Universal Robots PolyScope program: _adminCG-AssembleAToB.urp

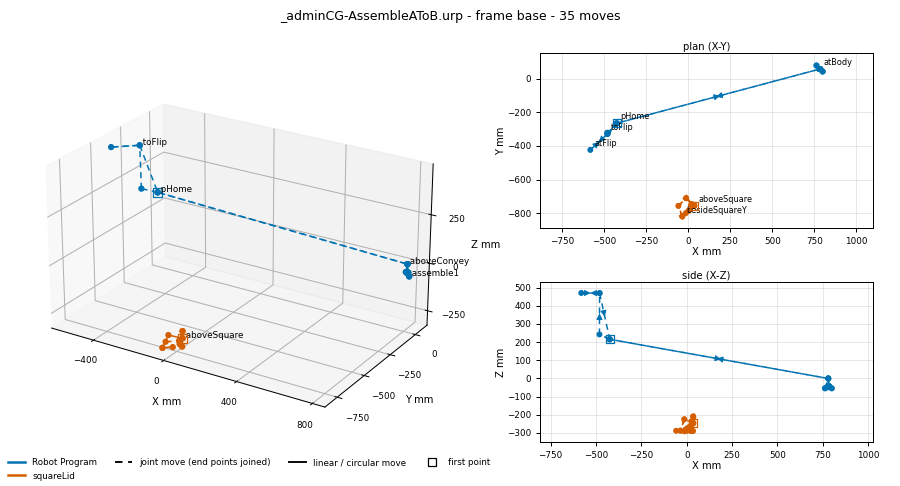
[picture p0: tool path of _adminCG-AssembleAToB.urp in frame base, 35 of 35 moves have a stored position in this frame; points joined in program order, loops and branches not executed]
Program _adminCG-AssembleAToB (installation=admin directory=/programs/WED_9AM createdIn=3.15.8.106339 lastSavedIn=3.15.8.106339 robotSerialNumber=2015350925)
Calibrated DH parameters: a=[0.000202, -0.047961, -0.392055, -0.000001, 0.000007, 0]; d=[0.089082, 828.736652, -823.627268, -4.999465, 0.094767, 0.082274]; alpha=[1.570325, 0.00051, -0.003464, 1.570175, -1.569769, 0]; deltaTheta=[0.000028, 1.457808, -1.502844, -6.238105, -6.283148, -0.000082]
Robot Program (runOnlyOnce=true)
  Set DigitalOutput pin=digital_out[0]; digitalValue=0
  MoveJ speed 60 deg/s, acceleration 80 deg/s^2 (useActiveTCP=true)
    Waypoint pHome: TCP in base x=-424.538 y=-265.05 z=215.597 mm, rx=-1.1995 ry=-2.8939 rz=-0.0048 rad; joints [224.997, -90.008, -90.005, -90.013, 89.259, -0.018] deg; flange x=-423.012 y=-266.393 z=431.487 mm, rx=-1.1995 ry=-2.8939 rz=-0.0048 rad
    Call _adminLinearIndex5
    Waypoint backUpFromFlip: TCP in base x=-481.215 y=-321.291 z=242.418 mm, rx=1.2187 ry=2.8869 rz=0.0126 rad; joints [224.559, -101.635, -73.028, -95.999, 90.041, 0.305] deg; flange x=-483.467 y=-322.229 z=458.304 mm, rx=1.2187 ry=2.8869 rz=0.0126 rad
  MoveJ speed 60 deg/s, acceleration 80 deg/s^2 (useActiveTCP=true)
    Waypoint toFlip: TCP in base x=-480.325 y=-329.398 z=470.329 mm, rx=0.0018 ry=0.0011 rz=-0.7778 rad; joints [225.307, -119.466, -107.5, -43.047, 269.775, 0.334] deg; flange x=-480.398 y=-328.953 z=254.429 mm, rx=0.0018 ry=0.0011 rz=-0.7778 rad
    Waypoint atFlip: TCP in base x=-581.465 y=-423.657 z=471.291 mm, rx=0.0073 ry=-0.0016 rz=-0.785 rad; joints [224.868, -133.376, -81.455, -55.525, 269.773, 0.333] deg; flange x=-580.559 y=-422.358 z=255.397 mm, rx=0.0073 ry=-0.0016 rz=-0.785 rad
    Set DigitalOutput pin=digital_out[0]; digitalValue=1
    Wait Sleep waitTime=1
    Set DigitalOutput pin=digital_out[2]; digitalValue=0
    Wait Sleep waitTime=1
    Waypoint toFlip: TCP in base x=-480.325 y=-329.398 z=470.329 mm, rx=0.0018 ry=0.0011 rz=-0.7778 rad; joints [225.307, -119.466, -107.5, -43.047, 269.775, 0.334] deg; flange x=-480.398 y=-328.953 z=254.429 mm, rx=0.0018 ry=0.0011 rz=-0.7778 rad
    Call _adminLinearIndex3
    Call squareLid
  MoveJ speed 60 deg/s, acceleration 80 deg/s^2 (useActiveTCP=true)
    Waypoint pHome: TCP in base x=-424.538 y=-265.05 z=215.597 mm, rx=-1.1995 ry=-2.8939 rz=-0.0048 rad; joints [224.997, -90.008, -90.005, -90.013, 89.259, -0.018] deg; flange x=-423.012 y=-266.393 z=431.487 mm, rx=-1.1995 ry=-2.8939 rz=-0.0048 rad
    Call _adminLinearIndex2
    Waypoint aboveConvey: TCP in base x=780.769 y=56.622 z=-0.465 mm, rx=1.1372 ry=-2.8707 rz=0.041 rad; joints [12.999, -136.609, -54.995, -81.263, 87.848, 59.736] deg; flange x=789.407 y=66.208 z=215.049 mm, rx=1.1372 ry=-2.8707 rz=0.041 rad
    Waypoint rotateConvey: TCP in base x=780.784 y=56.567 z=-0.471 mm, rx=2.895 ry=1.1467 rz=-0.0834 rad; joints [12.996, -136.61, -54.995, -81.26, 87.846, 239.737] deg; flange x=789.416 y=66.159 z=215.043 mm, rx=2.895 ry=1.1467 rz=-0.0834 rad
    Waypoint atBody: TCP in base x=780.781 y=56.499 z=-48.623 mm, rx=2.895 ry=1.1466 rz=-0.0836 rad; joints [12.996, -138.549, -58.718, -75.603, 87.846, 239.721] deg; flange x=789.426 y=66.117 z=166.89 mm, rx=2.895 ry=1.1466 rz=-0.0836 rad
    Wait Sleep waitTime=1
    Set DigitalOutput pin=digital_out[0]; digitalValue=0
    Wait Sleep waitTime=1
    Waypoint aboveConvey: TCP in base x=780.769 y=56.622 z=-0.465 mm, rx=1.1372 ry=-2.8707 rz=0.041 rad; joints [12.999, -136.609, -54.995, -81.263, 87.848, 59.736] deg; flange x=789.407 y=66.208 z=215.049 mm, rx=1.1372 ry=-2.8707 rz=0.041 rad
    Set DigitalOutput pin=digital_out[0]; digitalValue=1
    Waypoint abovePress: TCP in base x=785.714 y=57.816 z=-43.706 mm, rx=1.1164 ry=-2.8991 rz=0.0376 rad; joints [12.888, -138.367, -58.524, -74.941, 88.163, 60.68] deg; flange x=790.834 y=65.386 z=172.001 mm, rx=1.1164 ry=-2.8991 rz=0.0376 rad
  If force()≤65 (checkContinuously=true)
    MoveL speed 50 mm/s, acceleration 100 mm/s^2 (useActiveTCP=true) feature=Base
      Waypoint assemble1: TCP in base x=799.867 y=42.231 z=-54.523 mm, rx=1.1163 ry=-2.8991 rz=0.0375 rad; joints [11.574, -140.879, -55.504, -75.412, 88.126, 59.369] deg; flange x=805.001 y=49.793 z=161.183 mm, rx=1.1163 ry=-2.8991 rz=0.0375 rad
  MoveJ speed 60 deg/s, acceleration 80 deg/s^2 (useActiveTCP=true)
    Waypoint abovePress: TCP in base x=785.714 y=57.816 z=-43.706 mm, rx=1.1164 ry=-2.8991 rz=0.0376 rad; joints [12.888, -138.367, -58.524, -74.941, 88.163, 60.68] deg; flange x=790.834 y=65.386 z=172.001 mm, rx=1.1164 ry=-2.8991 rz=0.0376 rad
  If force()≤65 (checkContinuously=true)
    MoveL speed 50 mm/s, acceleration 100 mm/s^2 (useActiveTCP=true) feature=Base
      Waypoint assemble2: TCP in base x=763.064 y=78.057 z=-54.537 mm, rx=1.1164 ry=-2.8989 rz=0.0377 rad; joints [14.737, -135.9, -64.716, -71.278, 88.219, 62.516] deg; flange x=768.213 y=85.654 z=161.168 mm, rx=1.1164 ry=-2.8989 rz=0.0377 rad
  MoveJ speed 60 deg/s, acceleration 80 deg/s^2 (useActiveTCP=true)
    Waypoint abovePress: TCP in base x=785.714 y=57.816 z=-43.706 mm, rx=1.1164 ry=-2.8991 rz=0.0376 rad; joints [12.888, -138.367, -58.524, -74.941, 88.163, 60.68] deg; flange x=790.834 y=65.386 z=172.001 mm, rx=1.1164 ry=-2.8991 rz=0.0376 rad
  If force()≤65 (checkContinuously=true)
    MoveL speed 50 mm/s, acceleration 100 mm/s^2 (useActiveTCP=true) feature=Base
      Waypoint assemble1: TCP in base x=799.867 y=42.231 z=-54.523 mm, rx=1.1163 ry=-2.8991 rz=0.0375 rad; joints [11.574, -140.879, -55.504, -75.412, 88.126, 59.369] deg; flange x=805.001 y=49.793 z=161.183 mm, rx=1.1163 ry=-2.8991 rz=0.0375 rad
  MoveJ speed 60 deg/s, acceleration 80 deg/s^2 (useActiveTCP=true)
    Waypoint abovePress: TCP in base x=785.714 y=57.816 z=-43.706 mm, rx=1.1164 ry=-2.8991 rz=0.0376 rad; joints [12.888, -138.367, -58.524, -74.941, 88.163, 60.68] deg; flange x=790.834 y=65.386 z=172.001 mm, rx=1.1164 ry=-2.8991 rz=0.0376 rad
  If force()≤65 (checkContinuously=true)
    MoveL speed 50 mm/s, acceleration 100 mm/s^2 (useActiveTCP=true) feature=Base
      Waypoint assemble2: TCP in base x=763.064 y=78.057 z=-54.537 mm, rx=1.1164 ry=-2.8989 rz=0.0377 rad; joints [14.737, -135.9, -64.716, -71.278, 88.219, 62.516] deg; flange x=768.213 y=85.654 z=161.168 mm, rx=1.1164 ry=-2.8989 rz=0.0377 rad
  Call _adminLinearIndex2
  MoveJ speed 60 deg/s, acceleration 80 deg/s^2 (useActiveTCP=true)
    Waypoint aboveConvey: TCP in base x=780.769 y=56.622 z=-0.465 mm, rx=1.1372 ry=-2.8707 rz=0.041 rad; joints [12.999, -136.609, -54.995, -81.263, 87.848, 59.736] deg; flange x=789.407 y=66.208 z=215.049 mm, rx=1.1372 ry=-2.8707 rz=0.041 rad
    Waypoint pHome: TCP in base x=-424.538 y=-265.05 z=215.597 mm, rx=-1.1995 ry=-2.8939 rz=-0.0048 rad; joints [224.997, -90.008, -90.005, -90.013, 89.259, -0.018] deg; flange x=-423.012 y=-266.393 z=431.487 mm, rx=-1.1995 ry=-2.8939 rz=-0.0048 rad
SubProgram -> _adminLinearIndex3
SubProgram -> _adminLinearIndex5
SubProgram -> squareLid
SubProgram -> _adminLinearIndex2
SubProgram _adminLinearIndex5 (keepSynchronizedWithDisk=false) programFile=/programs/me345_admin/_adminLinearIndex5.urp
  Folder Move_linear_slide_Index5
    var_1 := False
    Loop While (checkContinuously=false) expression=var_1≟ False
      var_1 := socket_open("10.241.34.48",4001)
    var_3 := 1
    Send := "s r0x24 21"
    Script: socket_send_string(Send)
    Script: socket_send_byte(13)
    Send_Reply := socket_read_string()
    Send := "s r0xca 240000"
    Script: socket_send_string(Send)
    Script: socket_send_byte(13)
    Send_Reply := socket_read_string()
    Send := "t 1"
    Script: socket_send_string(Send)
    Script: socket_send_byte(13)
    Send_Reply := socket_read_string()
    Loop While (checkContinuously=false) expression=var_3≠0
      Send := "g r0xA0"
      Script: socket_send_string(Send)
      Script: socket_send_byte(13)
      var_3 := socket_get_var("v")
      Wait Sleep waitTime=0.1
    Script: socket_close()
    Script: sync()
SubProgram _adminLinearIndex3 (keepSynchronizedWithDisk=false) programFile=/programs/me345_admin/_adminLinearIndex3.urp
  Folder Move_linear_slide_Index3
    var_1 := False
    Loop While (checkContinuously=false) expression=var_1≟ False
      var_1 := socket_open("10.241.34.48",4001)
    var_3 := 1
    Send := "s r0x24 21"
    Script: socket_send_string(Send)
    Script: socket_send_byte(13)
    Send_Reply := socket_read_string()
    Send := "s r0xca 112778"
    Script: socket_send_string(Send)
    Script: socket_send_byte(13)
    Send_Reply := socket_read_string()
    Send := "t 1"
    Script: socket_send_string(Send)
    Script: socket_send_byte(13)
    Send_Reply := socket_read_string()
    Loop While (checkContinuously=false) expression=var_3≠0
      Send := "g r0xA0"
      Script: socket_send_string(Send)
      Script: socket_send_byte(13)
      var_3 := socket_get_var("v")
      Wait Sleep waitTime=0.1
    Script: socket_close()
    Script: sync()
SubProgram squareLid (keepSynchronizedWithDisk=false) programFile=/programs/WED_9AM/squareLid.urp
  MoveJ speed 60 deg/s, acceleration 80 deg/s^2 (useActiveTCP=true)
    Waypoint aboveSquare: TCP in base x=36.387 y=-754.554 z=-247.163 mm, rx=1.2016 ry=2.8994 rz=-0.0037 rad; joints [281.141, -148.015, -74.126, -47.712, 89.943, 55.968] deg; flange x=35.974 y=-753.836 z=-31.264 mm, rx=1.2016 ry=2.8994 rz=-0.0037 rad
  MoveL speed 250 mm/s, acceleration 1200 mm/s^2 (useActiveTCP=true) feature=Base
    Waypoint atSquare: TCP in base x=27.975 y=-754.016 z=-286.557 mm, rx=1.2021 ry=2.8995 rz=-0.0036 rad; joints [280.522, -151.75, -73.506, -44.611, 89.942, 55.355] deg; flange x=27.617 y=-753.337 z=-70.659 mm, rx=1.2021 ry=2.8995 rz=-0.0036 rad
    Set DigitalOutput pin=digital_out[0]; digitalValue=0
    Wait Sleep waitTime=1
    Waypoint aboveSquare: TCP in base x=36.387 y=-754.554 z=-247.163 mm, rx=1.2016 ry=2.8994 rz=-0.0037 rad; joints [281.141, -148.015, -74.126, -47.712, 89.943, 55.968] deg; flange x=35.974 y=-753.836 z=-31.264 mm, rx=1.2016 ry=2.8994 rz=-0.0037 rad
    Waypoint NextToSquare: TCP in base x=-13.128 y=-799.041 z=-224.591 mm, rx=1.2019 ry=2.8993 rz=-0.0035 rad; joints [276.969, -151.009, -63.364, -55.49, 89.947, 51.825] deg; flange x=-13.559 y=-798.339 z=-8.693 mm, rx=1.2019 ry=2.8993 rz=-0.0035 rad
    Set DigitalOutput pin=digital_out[0]; digitalValue=1
    Wait Sleep waitTime=0.5
  MoveJ speed 180 deg/s, acceleration 100 deg/s^2 (useActiveTCP=true)
    Waypoint besideSquareY: TCP in base x=-34.238 y=-818.585 z=-288.276 mm, rx=1.2017 ry=2.8994 rz=-0.0033 rad; joints [275.321, -159.315, -56.448, -54.11, 89.96, 50.165] deg; flange x=-34.671 y=-817.911 z=-72.378 mm, rx=1.2017 ry=2.8994 rz=-0.0033 rad
  Wait Sleep waitTime=0.1
  MoveL speed 30 mm/s, acceleration 30 mm/s^2 (useActiveTCP=true) feature=Base
    If force()≤45 (checkContinuously=true)
      Waypoint atSquareY_1: TCP in base x=1.543 y=-785.766 z=-288.889 mm, rx=1.2019 ry=2.899 rz=-0.0034 rad; joints [278.16, -155.287, -65.735, -48.838, 89.971, 53.003] deg; flange x=1.069 y=-785.066 z=-72.991 mm, rx=1.2019 ry=2.899 rz=-0.0034 rad
    Wait Sleep waitTime=0.5
  MoveJ speed 180 deg/s, acceleration 100 deg/s^2 (useActiveTCP=true)
    Waypoint besideSquareY: TCP in base x=-34.238 y=-818.585 z=-288.276 mm, rx=1.2017 ry=2.8994 rz=-0.0033 rad; joints [275.321, -159.315, -56.448, -54.11, 89.96, 50.165] deg; flange x=-34.671 y=-817.911 z=-72.378 mm, rx=1.2017 ry=2.8994 rz=-0.0033 rad
    Waypoint linkingMove: motionParameters(blendRadius=0.005); TCP in base x=-58.166 y=-756.622 z=-289.108 mm, rx=1.2018 ry=2.8995 rz=-0.0034 rad; joints [273.941, -152.445, -72.394, -45.037, 89.973, 48.766] deg; flange x=-58.56 y=-755.949 z=-73.21 mm, rx=1.2018 ry=2.8995 rz=-0.0034 rad
    Waypoint besideSquareX: TCP in base x=-11.874 y=-710.677 z=-291.242 mm, rx=1.2017 ry=2.8995 rz=-0.0033 rad; joints [277.95, -148.186, -83.128, -38.559, 89.981, 52.757] deg; flange x=-12.29 y=-710.014 z=-75.343 mm, rx=1.2017 ry=2.8995 rz=-0.0033 rad
  Wait Sleep waitTime=0.1
  MoveL speed 30 mm/s, acceleration 30 mm/s^2 (useActiveTCP=true) feature=Base
    If force()≤45 (checkContinuously=true)
      Waypoint atSquareX_1: TCP in base x=21.957 y=-744.876 z=-290.622 mm, rx=1.2021 ry=2.8994 rz=-0.0033 rad; joints [280.187, -151.247, -75.553, -43.073, 89.958, 55.016] deg; flange x=21.56 y=-744.226 z=-74.723 mm, rx=1.2021 ry=2.8994 rz=-0.0033 rad
    Wait Sleep waitTime=0.5
  MoveJ speed 60 deg/s, acceleration 80 deg/s^2 (useActiveTCP=true)
    Waypoint besideSquareX: TCP in base x=-11.874 y=-710.677 z=-291.242 mm, rx=1.2017 ry=2.8995 rz=-0.0033 rad; joints [277.95, -148.186, -83.128, -38.559, 89.981, 52.757] deg; flange x=-12.29 y=-710.014 z=-75.343 mm, rx=1.2017 ry=2.8995 rz=-0.0033 rad
    Waypoint aboveSquare2: TCP in base x=36.038 y=-754.121 z=-209.989 mm, rx=1.2012 ry=2.8998 rz=-0.0034 rad; joints [281.12, -144.584, -74.474, -50.811, 89.931, 55.933] deg; flange x=35.647 y=-753.459 z=5.91 mm, rx=1.2012 ry=2.8998 rz=-0.0034 rad
    Set DigitalOutput pin=digital_out[0]; digitalValue=0
    Wait Sleep waitTime=1
  MoveL speed 250 mm/s, acceleration 1200 mm/s^2 (useActiveTCP=true) feature=Base
    Waypoint atSquare2: TCP in base x=34.929 y=-756.694 z=-290.333 mm, rx=1.2013 ry=2.8997 rz=-0.0033 rad; joints [281.004, -152.426, -72.693, -44.749, 89.951, 55.806] deg; flange x=34.531 y=-756.032 z=-74.435 mm, rx=1.2013 ry=2.8997 rz=-0.0033 rad
    Set DigitalOutput pin=digital_out[0]; digitalValue=1
    Wait Sleep waitTime=1
    Waypoint easeout: TCP in base x=16.999 y=-751.256 z=-283.255 mm, rx=1.2013 ry=2.8997 rz=-0.0032 rad; joints [279.722, -151.117, -74.307, -44.451, 89.958, 54.524] deg; flange x=16.598 y=-750.614 z=-67.356 mm, rx=1.2013 ry=2.8997 rz=-0.0032 rad
    Waypoint aboveSquare2: TCP in base x=36.038 y=-754.121 z=-209.989 mm, rx=1.2012 ry=2.8998 rz=-0.0034 rad; joints [281.12, -144.584, -74.474, -50.811, 89.931, 55.933] deg; flange x=35.647 y=-753.459 z=5.91 mm, rx=1.2012 ry=2.8998 rz=-0.0034 rad
SubProgram _adminLinearIndex2 (keepSynchronizedWithDisk=false) programFile=/programs/me345_admin/_adminLinearIndex2.urp
  Folder Move_linear_slide_Index2
    var_1 := False
    Loop While (checkContinuously=false) expression=var_1≟ False
      var_1 := socket_open("10.241.34.48",4001)
    var_3 := 1
    Send := "s r0x24 21"
    Script: socket_send_string(Send)
    Script: socket_send_byte(13)
    Send_Reply := socket_read_string()
    Send := "s r0xca 51968"
    Script: socket_send_string(Send)
    Script: socket_send_byte(13)
    Send_Reply := socket_read_string()
    Send := "t 1"
    Script: socket_send_string(Send)
    Script: socket_send_byte(13)
    Send_Reply := socket_read_string()
    Loop While (checkContinuously=false) expression=var_3≠0
      Send := "g r0xA0"
      Script: socket_send_string(Send)
      Script: socket_send_byte(13)
      var_3 := socket_get_var("v")
      Wait Sleep waitTime=0.1
    Script: socket_close()
    Script: sync()
